// TIA Portal V16 export
// export: Created 2023-08-28T09:37:55.4310904Z, ExportSetting WithDefaults, DisplayName Totally Integrated Automation Portal, DisplayVersion V16 Update 6, DisplayName TIA Portal Version Control Interface, DisplayVersion V16 Update 2, DisplayName TIA Portal Openness, DisplayVersion V16 Update 6, DisplayName STEP 7 Professional, DisplayVersion V16 Update 6, DisplayName STEP 7 Safety, DisplayVersion V16, DisplayName WinCC Advanced, DisplayVersion V16 Update 6
VAR_GLOBAL   // PLC tag table "Tag VLV01"
   Valve_Bit_K AT %M20.6 : Bool;   // Bit-6 kasowanie alarmu
   IN_STAT_Velv01 AT %MW20 : Word;   // Wejściowe słowo statusu napędu
   "Valve_Bit_A/R" AT %M20.7 : Bool;   // Bit trybu pracy napędu
   Valve_Bit_C AT %M20.5 : Bool;   // Rozkaz zamykania
   Valve_Bit_Open AT %M20.4 : Bool;   // Rozkaz otwieranie
   Valve_BIT_A AT %M20.0 : Bool;   // Bit gotowośći / awarii
   Byte_Wekt_Valve01 AT %MW24 : Word;   // Out- słowo wektora napędu
   "Bit_0-Wekt_Valve01" AT %M21.0 : Bool;   // Bit Alarm/Gotowość (Alarm-=1, gotowość=0)
   "Bit_1-Wekt_Valve01" AT %M21.1 : Bool;   // Bit potwierdzenia otwarcia
   "Bit_2-Wekt_Valve01" AT %M21.2 : Bool;   // Bit wyboru trybu Zdalne=1 Remontowe=0
   "Bit_3-Wek_Valve01" AT %M21.3 : Bool;   // Bit potwierdzenia zamknięcia
   "Bit_4-Wek_Valve01" AT %M21.4 : Bool;   // Bit rozkazu na otwieranie
   "Bit_5-Wekt-Valve01" AT %M21.5 : Bool;   // Bit rozkazu na zamykanie
   "Bit_6-Wekt-Valve01" AT %M21.6 : Bool;   // Bit kasowania
   "Bit_7-Wekt-Valve01" AT %M21.7 : Bool;   // Bit rodzaju sterowania aut =1 /manual= 0
   Byte_Wekt_Valve01_L AT %MB21 : Byte;   // Lewy byte wektora napędu
   Byte_Wekt_Valve01_R AT %MB20 : Byte;   // Prawy byte wektora napędu
   ByteH_Status_P1 AT %MB60 : Byte;   // status napędu
END_VAR
